// TIA Portal V20 export
// export: Created 2026-07-12T13:33:04.7738954Z, ExportSetting WithDefaults, DisplayName Totally Integrated Automation Portal, DisplayVersion V20 Update 4, DisplayName TIA Portal Openness, DisplayVersion V20 Update 4, DisplayName TIA Portal Version Control Interface, DisplayVersion V20 Update 4, DisplayName STEP 7 Professional, DisplayVersion V20 Update 4, DisplayName STEP 7 Safety, DisplayVersion V20 Update 2, DisplayName WinCC Basic/Comfort/Advanced, DisplayVersion V20 Update 4, DisplayName WinCC Unified, DisplayVersion V20 Update 4
DATA_BLOCK "DB_DataHandler"   // DB4
{ S7_Optimized_Access := 'FALSE' }
VERSION : 0.1
// stored: AutoNumber true, IsOnlyStoredInLoadMemory false, IsWriteProtectedInAS false
   VAR RETAIN
      ProfileSelectrion : Word;
      ProfileRead : Word;
      Exception : Bool;
      ProfileEn : Bool;
      CountBuffer : Array[0..3] of Word;
      CutData : Array[0..3] of "UDT_CutData";
      SawDone { S7_SetPoint := 'True'} : Bool;
   END_VAR
BEGIN
END_DATA_BLOCK
